// TIA Portal V21 export
VAR_GLOBAL   // PLC tag table "KAllRicetta"
END_VAR
